// TwinCAT 3 PLC project PLC
// ProgramVersion: 3.1.4026.24
// libraries:
//   Tc2_EtherCAT, * (Beckhoff Automation GmbH)
//   Tc2_Standard, * (Beckhoff Automation GmbH)
//   Tc2_System, * (Beckhoff Automation GmbH)
//   Tc3_EventLogger, * (Beckhoff Automation GmbH)
//   Tc3_PackML_V3, * (Beckhoff Automation GmbH)
// project tree:
//   Machine Module/ MachineModule.TcPOU
//   / MAIN.TcPOU, PlcTask.TcTTO
//   Visu %28Local Debug Only%29/ GlobalTextList.TcGTLO (not stored), Visualization Manager.TcVMO (not stored), V_Main.TcVIS (not stored)
//   Visu %28Local Debug Only%29/User Controls/ V_PackMLModule.TcVIS (not stored)
//   _Internal/PackML Module %28Base%29/ I_PackML_Module.TcIO (not stored), NextAvailablePackMLCommands.TcPOU (not stored), PackMLModule.TcPOU (not stored), PackMLStatemachine_HMI.TcPOU (not stored), ST_PackMLStatemachine_HMI.TcDUT (not stored)
//   _Internal/Steps/ NextMinorStep.TcPOU, NextStep.TcPOU, SetStep.TcPOU
//   _Internal/Trace/ AdsLogger.TcPOU, GvlTrace.TcGVL, TcEventLogger.TcPOU, Trace.TcPOU, USINT_To_TcEventSeverity.TcPOU (not stored)
//   _Internal/Trace/DUT/ TcEventSeverityExt.TcDUT (not stored)
//   _Internal/Trace/Interface/ I_Base.TcIO, I_ContainTraceArgument.TcIO, I_ContainTracePublisher.TcIO, I_ToString.TcIO, I_Trace.TcIO (not stored), I_TraceArgument.TcIO, I_TraceInstanceLogger.TcIO, I_TraceLogger.TcIO, I_TraceMessageInfo.TcIO, I_TracePublisher.TcIO, I_TraceSourceInfo.TcIO
// real-time tasks:
//   TASK PlcTask: cycle T#10ms, priority 20, ADS port 350

CONFIGURATION PLC
    RESOURCE PLC ON TwinCAT3
        TASK PlcTask(INTERVAL := T#10ms, PRIORITY := 20);
        PROGRAM MAIN WITH PlcTask : MAIN;
    END_RESOURCE
END_CONFIGURATION

// ---- _Internal/Trace/GvlTrace.TcGVL
VAR_GLOBAL
    EnableAdsLogger : BOOL := TRUE;
    EnableTcEventLogging : BOOL := FALSE;
    TraceLevel : TcEventSeverityExt := TcEventSeverityExt.Verbose;
	Trace : Trace<10> := (TraceLevel := TraceLevel);
	TcEventLogger : TcEventLogger(Trace);
	AdsLogger : AdsLogger(Trace);
END_VAR

// ---- _Internal/Trace/Interface/I_Base.TcIO
INTERFACE I_Base EXTENDS __SYSTEM.IQueryInterface

END_INTERFACE

// ---- _Internal/Trace/Interface/I_ContainTraceArgument.TcIO
INTERFACE I_ContainTraceArgument EXTENDS I_Base

{attribute 'monitoring' := 'call'}
PROPERTY Arguments : I_TraceArgument
GET
END_GET
END_PROPERTY

END_INTERFACE

// ---- _Internal/Trace/Interface/I_ContainTracePublisher.TcIO
INTERFACE I_ContainTracePublisher EXTENDS I_Base

PROPERTY Publisher : I_TracePublisher
GET
END_GET
END_PROPERTY

END_INTERFACE

// ---- _Internal/Trace/Interface/I_ToString.TcIO
INTERFACE I_ToString EXTENDS I_Base

METHOD ToString : T_MaxString
VAR_INPUT
END_VAR
END_METHOD

END_INTERFACE

// ---- _Internal/Trace/Interface/I_TraceArgument.TcIO
INTERFACE I_TraceArgument EXTENDS I_ToString

END_INTERFACE

// ---- _Internal/Trace/Interface/I_TraceInstanceLogger.TcIO
INTERFACE I_TraceInstanceLogger EXTENDS I_Base

METHOD LogMessageInstance
VAR_INPUT
	SourceInfo	: I_TraceSourceInfo;
	MessageInfo : I_TraceMessageInfo;
	Arguments	: I_TraceArgument := 0;
END_VAR
END_METHOD

END_INTERFACE

// ---- _Internal/Trace/Interface/I_TraceLogger.TcIO
INTERFACE I_TraceLogger EXTENDS I_Base

METHOD LogMessage
VAR_INPUT
	Key		  : T_MaxString;
	Value	  : T_MaxString;
	SourceId  : UDINT := 0;
	TimeStamp : ULINT := 0;
	MessageId : UDINT := 1;
	Severity  : USINT := 1;
END_VAR
END_METHOD

END_INTERFACE

// ---- _Internal/Trace/Interface/I_TraceMessageInfo.TcIO
INTERFACE I_TraceMessageInfo EXTENDS I_Base

{attribute 'monitoring':='call'}
PROPERTY Message : T_MaxString
GET
END_GET
END_PROPERTY

{attribute 'monitoring':='call'}
PROPERTY MessageId : UDINT
GET
END_GET
END_PROPERTY

{attribute 'monitoring':='call'}
PROPERTY Severity : USINT
GET
END_GET
END_PROPERTY

END_INTERFACE

// ---- _Internal/Trace/Interface/I_TracePublisher.TcIO
INTERFACE I_TracePublisher

METHOD Subscribe
VAR_INPUT
	Logger : I_TraceLogger;
END_VAR
END_METHOD

METHOD Unsubscribe
VAR_INPUT
	Logger : I_TraceLogger;
END_VAR
END_METHOD

END_INTERFACE

// ---- _Internal/Trace/Interface/I_TraceSourceInfo.TcIO
INTERFACE I_TraceSourceInfo EXTENDS I_Base

{attribute 'monitoring':='call'}
PROPERTY SourceId : UDINT
GET
END_GET
END_PROPERTY

{attribute 'monitoring':='call'}
PROPERTY SourceName : T_MaxString
GET
END_GET
END_PROPERTY

{attribute 'monitoring':='call'}
PROPERTY TimeStamp : ULINT
GET
END_GET
END_PROPERTY

END_INTERFACE

// ---- MAIN.TcPOU
PROGRAM MAIN
VAR
    Machine : MachineModule('Machine 1');
    Machine_HMI : PackMLStatemachine_HMI('Machine 1 HMI', Machine);
END_VAR

Machine.CyclicLogic();
Machine_HMI.CyclicLogic();

END_PROGRAM

// ---- Machine Module/MachineModule.TcPOU
FUNCTION_BLOCK MachineModule EXTENDS PackMLModule
VAR
    Initialized : BOOL;
    SimulatedError : BOOL;
    {attribute 'OPC.UA.DA' := '1'}
	_PackTags : ST_PMLV2022;
END_VAR

METHOD Aborting : BOOL
Aborting := TRUE;
END_METHOD

METHOD Clearing : BOOL
SimulatedError := FALSE;
Clearing := TRUE;
END_METHOD

METHOD CyclicLogic
VAR_INST
    ErrorRT : R_TRIG;
END_VAR
IF NOT Initialized THEN
    Initialize();
    RETURN;
END_IF

SUPER^.CyclicLogic();
UpdateTimers();

ErrorRT(CLK := SimulatedError);
IF ErrorRT.Q THEN
    Trace.Error(Name, 'Error occured -> Abort Statemachine');
    ChangeState(E_PMLCommand.Abort);
END_IF
END_METHOD

METHOD Execute : BOOL
END_METHOD

METHOD Initialize
VAR_INST
	UnitModeConfig : FB_PMLUnitModeConfig;
END_VAR
CASE SequenceState OF
	0:
		UnitModeConfig(eMode						  := E_PMLProtectedUnitMode.Production,
					   sName						  := 'Mode Production',
					   bDisableClearing				  := FALSE,
					   bDisableStarting				  := FALSE,
					   bDisableSuspended			  := FALSE,
					   bDisableStopping				  := FALSE,
					   bDisableAborting				  := FALSE,
					   bDisableHolding				  := FALSE,
					   bDisableHeld					  := FALSE,
					   bDisableUnholding			  := FALSE,
					   bDisableSuspending			  := FALSE,
					   bDisableUnsuspending			  := FALSE,
					   bDisableResetting			  := FALSE,
					   bDisableIdle					  := FALSE,
					   bDisableCompleting			  := FALSE,
					   bDisableComplete				  := FALSE,
					   bEnableUnitModeChangeStopped	  := TRUE,
					   bEnableUnitModeChangeIdle	  := FALSE,
					   bEnableUnitModeChangeSuspended := FALSE,
					   bEnableUnitModeChangeExecute	  := FALSE,
					   bEnableUnitModeChangeAborted	  := TRUE,
					   bEnableUnitModeChangeHeld	  := FALSE,
					   bEnableUnitModeChangeComplete  := FALSE,
					   bError						  =>,
					   nErrorId						  =>);

		UnitModeConfig(eMode						  := E_PMLProtectedUnitMode.Maintenance,
					   sName						  := 'Mode Maintenance',
					   bDisableClearing				  := FALSE,
					   bDisableStarting				  := FALSE,
					   bDisableSuspended			  := FALSE,
					   bDisableStopping				  := FALSE,
					   bDisableAborting				  := FALSE,
					   bDisableHolding				  := FALSE,
					   bDisableHeld					  := FALSE,
					   bDisableUnholding			  := FALSE,
					   bDisableSuspending			  := FALSE,
					   bDisableUnsuspending			  := FALSE,
					   bDisableResetting			  := FALSE,
					   bDisableIdle					  := FALSE,
					   bDisableCompleting			  := FALSE,
					   bDisableComplete				  := FALSE,
					   bEnableUnitModeChangeStopped	  := TRUE,
					   bEnableUnitModeChangeIdle	  := FALSE,
					   bEnableUnitModeChangeSuspended := FALSE,
					   bEnableUnitModeChangeExecute	  := FALSE,
					   bEnableUnitModeChangeAborted	  := TRUE,
					   bEnableUnitModeChangeHeld	  := FALSE,
					   bEnableUnitModeChangeComplete  := FALSE,
					   bError						  =>,
					   nErrorId						  =>);

		UnitModeConfig(eMode						  := E_PMLProtectedUnitMode.Manual,
					   sName						  := 'Mode Manual',
					   bDisableClearing				  := FALSE,
					   bDisableStarting				  := FALSE,
					   bDisableSuspended			  := FALSE,
					   bDisableStopping				  := FALSE,
					   bDisableAborting				  := FALSE,
					   bDisableHolding				  := FALSE,
					   bDisableHeld					  := FALSE,
					   bDisableUnholding			  := FALSE,
					   bDisableSuspending			  := FALSE,
					   bDisableUnsuspending			  := FALSE,
					   bDisableResetting			  := FALSE,
					   bDisableIdle					  := FALSE,
					   bDisableCompleting			  := FALSE,
					   bDisableComplete				  := FALSE,
					   bEnableUnitModeChangeStopped	  := TRUE,
					   bEnableUnitModeChangeIdle	  := FALSE,
					   bEnableUnitModeChangeSuspended := FALSE,
					   bEnableUnitModeChangeExecute	  := FALSE,
					   bEnableUnitModeChangeAborted	  := TRUE,
					   bEnableUnitModeChangeHeld	  := FALSE,
					   bEnableUnitModeChangeComplete  := FALSE,
					   bError						  =>,
					   nErrorId						  =>);

		NextStep(SequenceState);

	10:
		Initialized := TRUE;
END_CASE
END_METHOD

METHOD Resetting : BOOL
Resetting := TRUE;
END_METHOD

METHOD Starting : BOOL
CASE CurrentMode OF
    E_PMLProtectedUnitMode.Production:
        CASE SequenceState OF 
            0:
                // Start Production Mode
                NextStep(SequenceState);
                
            10:
                // State completed -> transition by setting state to TRUE
                Starting := TRUE;
            
        END_CASE
    
    E_PMLProtectedUnitMode.Maintenance:
        Starting := TRUE;
      
ELSE
    Starting := TRUE;
END_CASE
END_METHOD

METHOD Stopping : BOOL
Stopping := TRUE;
END_METHOD

METHOD UpdateTimers
VAR
	CurrentTime	 : T_DCTIME64;
	TimeToUpdate : LREAL;
END_VAR

VAR_INST
	LastTime  : T_DCTIME64 := F_GetActualDcTime64();
	LastState : DINT;
	LastMode  : DINT;
END_VAR
IF _PackTags.Status.StateCurrent <> LastState THEN
	MEMSET(ADR(_PackTags.Admin.StateTimeCurrent), 0, SIZEOF(_PackTags.Admin.StateTimeCurrent));
	LastState := _PackTags.Status.StateCurrent;
END_IF

IF _PackTags.Status.UnitModeCurrent <> LastMode THEN
	MEMSET(ADR(_PackTags.Admin.ModeTimeCurrent), 0, SIZEOF(_PackTags.Admin.ModeTimeCurrent));
	LastMode := _PackTags.Status.UnitModeCurrent;
END_IF

CurrentTime := F_GetActualDcTime64();
IF LastTime <> 0 THEN
	TimeToUpdate := ULINT_TO_LREAL(CurrentTime - LastTime) / 1_000_000_000.0;
END_IF
END_METHOD

END_FUNCTION_BLOCK

// ---- _Internal/Trace/Trace.TcPOU
FUNCTION_BLOCK Trace
VAR_GENERIC CONSTANT
	MaxCount : UDINT := 10;
END_VAR IMPLEMENTS I_TracePublisher, I_Trace, I_TraceLogger
VAR
	Loggers : ARRAY[0..MaxCount] OF I_TraceLogger;
	_TraceLevel : TcEventSeverityExt := TcEventSeverityExt.Warning;
END_VAR

METHOD Critical
VAR_INPUT
	Source	  : T_MaxString;
	Message	  : T_MaxString;
END_VAR
VAR
	i : UDINT;
END_VAR
FOR i := 0 TO MaxCount DO
	IF Loggers[i] <> 0 AND_THEN _TraceLevel < 5 THEN
		Loggers[i].LogMessage(Source,
							  Message,
							  0,
							  0,
							  1,
							  4);
	END_IF
END_FOR
END_METHOD

METHOD Error
VAR_INPUT
	Source	  : T_MaxString;
	Message	  : T_MaxString;
END_VAR
VAR
	i : UDINT;
END_VAR
FOR i := 0 TO MaxCount DO
	IF Loggers[i] <> 0 AND_THEN _TraceLevel < 4 THEN
		Loggers[i].LogMessage(Source,
							  Message,
							  0,
							  0,
							  1,
							  3);
	END_IF
END_FOR
END_METHOD

METHOD Info
VAR_INPUT
	Source	  : T_MaxString;
	Message	  : T_MaxString;
END_VAR
VAR
	i : UDINT;
END_VAR
FOR i := 0 TO MaxCount DO
	IF Loggers[i] <> 0 AND_THEN _TraceLevel < 2 THEN
		Loggers[i].LogMessage(Source,
							  Message,
							  0,
							  0,
							  1,
							  1);
	END_IF
END_FOR
END_METHOD

METHOD LogMessage
VAR_INPUT
	Key		  : T_MaxString;
	Value	  : T_MaxString;
	SourceId  : UDINT := 0;
	TimeStamp : ULINT := 0;
	MessageId : UDINT := 1;
	Severity  : USINT := 1;
END_VAR

VAR
	i : UDINT;
END_VAR
FOR i := 0 TO MaxCount DO
	IF Loggers[i] <> 0 THEN
		Loggers[i].LogMessage(Key,
							  Value,
							  SourceId,
							  TimeStamp,
							  MessageId,
							  Severity);
	END_IF
END_FOR
END_METHOD

METHOD Subscribe
VAR_INPUT
	Logger : I_TraceLogger;
END_VAR

VAR
	i : UDINT;
END_VAR
FOR i := 0 TO 10 DO
	IF Loggers[i] = 0 THEN
		Loggers[i] := Logger;
		EXIT;
	END_IF
END_FOR
END_METHOD

PROPERTY TraceLevel : TcEventSeverityExt
GET
TraceLevel := _TraceLevel;
END_GET
SET
_TraceLevel := TraceLevel;
END_SET
END_PROPERTY

METHOD Unsubscribe
VAR_INPUT
	Logger : I_TraceLogger;
END_VAR

VAR
	i : UDINT;
END_VAR
FOR i := 0 TO 10 DO
	IF Loggers[i] = Logger THEN
		Loggers[i] := 0;
		EXIT;
	END_IF
END_FOR
END_METHOD

METHOD Verbose
VAR_INPUT
	Source	  : T_MaxString;
	Message	  : T_MaxString;
END_VAR
VAR
	i : UDINT;
END_VAR
FOR i := 0 TO MaxCount DO
	IF Loggers[i] <> 0 AND_THEN _TraceLevel = 0 THEN
		Loggers[i].LogMessage(Source,
							  Message,
							  0,
							  0,
							  1,
							  0);
	END_IF
END_FOR
END_METHOD

METHOD Warning
VAR_INPUT
	Source	  : T_MaxString;
	Message	  : T_MaxString;
END_VAR
VAR
	i : UDINT;
END_VAR
FOR i := 0 TO MaxCount DO
	IF Loggers[i] <> 0 AND_THEN _TraceLevel < 3 THEN
		Loggers[i].LogMessage(Source,
							  Message,
							  0,
							  0,
							  1,
							  2);
	END_IF
END_FOR
END_METHOD

END_FUNCTION_BLOCK

// ---- _Internal/Steps/NextStep.TcPOU
FUNCTION NextStep : UDINT
VAR_IN_OUT
	StateVar : UDINT;
END_VAR

NextStep := StateVar := ((StateVar / 10) * 10) + 10;

END_FUNCTION

// ---- _Internal/Trace/TcEventLogger.TcPOU
FUNCTION_BLOCK TcEventLogger IMPLEMENTS I_TraceLogger
VAR
	MessagesThisScan : DINT;
	Message			 : FB_TcMessage;
	Source			 : FB_TcSourceInfo;
	CurrentCycle	 : UDINT;
END_VAR

//FB_Init is always available implicitly and it is used primarily for initialization.

//The return value is not evaluated. For a specific influence, you can also declare the

//methods explicitly and provide additional code there with the standard initialization

//code. You can evaluate the return value.
METHOD FB_Init : BOOL
VAR_INPUT
	bInitRetains   : BOOL; // TRUE: the retain variables are initialized (reset warm / reset cold)
	bInCopyCode	   : BOOL; // TRUE: the instance will be copied to the copy code afterward (online change)   
	TracePublisher : I_TracePublisher;
END_VAR
IF EnableTcEventLogging THEN
	TracePublisher.Subscribe(THIS^);
END_IF
END_METHOD

METHOD LogMessage
VAR_INPUT
	Key		  : T_MaxString;
	Value	  : T_MaxString;
	SourceId  : UDINT := 0;
	TimeStamp : ULINT := 0;
	MessageId : UDINT := 1;
	Severity  : USINT := 1;
END_VAR
IF GETCURTASKINDEXEX() > 0 THEN
    IF TwinCAT_SystemInfoVarList._TaskInfo[GETCURTASKINDEXEX()].CycleCount <> CurrentCycle THEN
        CurrentCycle	 := TwinCAT_SystemInfoVarList._TaskInfo[GETCURTASKINDEXEX()].CycleCount;
        MessagesThisScan := 0;
    END_IF
    
    IF NOT (MessagesThisScan < TO_DINT(TwinCAT_SystemInfoVarList._TaskInfo[GETCURTASKINDEXEX()].CycleTime / 2000)) THEN
        RETURN;
    END_IF
END_IF
  
Source.sName := Key;
Source.nId	 := SourceId;
Message.Create(eventClass	:= TC_EVENT_CLASSES.Trace,
			   nEventId		:= MessageId,
			   eSeverity	:= USINT_To_TcEventSeverity(Severity),
			   ipSourceInfo := Source);

Message.ipArguments.Clear().AddString(Value);
Message.Send(TimeStamp);
Message.Release();
Source.Clear();
MessagesThisScan := MessagesThisScan + 1;
END_METHOD

END_FUNCTION_BLOCK

// ---- _Internal/Trace/AdsLogger.TcPOU
FUNCTION_BLOCK AdsLogger IMPLEMENTS I_TraceLogger
VAR
	MessagesThisScan : DINT;
	CurrentCycle	 : UDINT;
END_VAR

//FB_Init is always available implicitly and it is used primarily for initialization.

//The return value is not evaluated. For a specific influence, you can also declare the

//methods explicitly and provide additional code there with the standard initialization

//code. You can evaluate the return value.
METHOD FB_Init : BOOL
VAR_INPUT
	bInitRetains   : BOOL; // TRUE: the retain variables are initialized (reset warm / reset cold)
	bInCopyCode	   : BOOL; // TRUE: the instance will be copied to the copy code afterward (online change)   
	TracePublisher : I_TracePublisher;
END_VAR
IF EnableAdsLogger THEN
	TracePublisher.Subscribe(THIS^);
END_IF
END_METHOD

METHOD LogMessage
VAR_INPUT
	Key		  : T_MaxString;
	Value	  : T_MaxString;
	SourceId  : UDINT := 0;
	TimeStamp : ULINT := 0;
	MessageId : UDINT := 1;
	Severity  : USINT := 1;
END_VAR
IF GETCURTASKINDEXEX() > 0 THEN
    IF TwinCAT_SystemInfoVarList._TaskInfo[GETCURTASKINDEXEX()].CycleCount <> CurrentCycle THEN
        CurrentCycle	 := TwinCAT_SystemInfoVarList._TaskInfo[GETCURTASKINDEXEX()].CycleCount;
        MessagesThisScan := 0;
    END_IF
    
    IF NOT (MessagesThisScan < TO_DINT(TwinCAT_SystemInfoVarList._TaskInfo[GETCURTASKINDEXEX()].CycleTime / 2000)) THEN
        RETURN;
    END_IF
END_IF


CASE Severity OF
	0, 1:
		ADSLOGSTR(ADSLOG_MSGTYPE_LOG OR ADSLOG_MSGTYPE_HINT, Concat(Value, ': %s'), Key);

	2:
		ADSLOGSTR(ADSLOG_MSGTYPE_LOG OR ADSLOG_MSGTYPE_WARN, Concat(Value, ': %s'), Key);

	3, 4:
		ADSLOGSTR(ADSLOG_MSGTYPE_LOG OR ADSLOG_MSGTYPE_ERROR, Concat(Value, ': %s'), Key);
END_CASE

MessagesThisScan := MessagesThisScan + 1;
END_METHOD

END_FUNCTION_BLOCK

// ---- _Internal/Steps/NextMinorStep.TcPOU
FUNCTION NextMinorStep : UDINT
VAR_IN_OUT
	StateVar : UDINT;
END_VAR

NextMinorStep := StateVar := StateVar + 1;

END_FUNCTION

// ---- _Internal/Steps/SetStep.TcPOU
FUNCTION SetStep : UDINT
VAR_IN_OUT
	StateVar : UDINT;
END_VAR

VAR_INPUT
	Step : UDINT;
END_VAR

SetStep := StateVar := Step;

END_FUNCTION
